TYPE ST_PendantControl :
STRUCT
	fTargetPosition : LREAL;
	fVelocity : LREAL := 100;
	fFwdLimit : LREAL;
	fBwdLimit : LREAL;
	fLocalModeSpeedOverride : LREAL;
END_STRUCT
END_TYPE

(* stored: Version 1.1.0.1, ProductVersion 3.1.4026.18
   DUT ST_PendantControl: Id {af3cd7ba-0cc2-4c79-b8f0-e738ae733380} *)
